FUNCTION_BLOCK MACH_CTL (* Cycle Control for a Machine with Fixed Tool *)
  (* Standard: 61499-1; Classification: Simulation; ApplicationDomain: Machining; Function: Drilling *)
  (* Version 0.2, 2004-10-20, JHC, Rockwell Automation, Changed algorithm to LD to recover from retracting fault. *)
  (* Version 0.1, 2004-04-05, JHC, Rockwell Automation, Corrected transition SPIN -> ADV *)
  (* Version 0.0, 2002-10-03, JHC, Rockwell Automation, Modified from DRILL_CTL. *)
  (* Compiler header: package fb.rt.mach; *)
  (* Compiler Java Sun JDK 1.4.2 *)
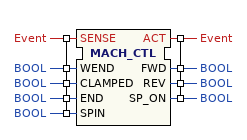
  EVENT_INPUT
    SENSE WITH WEND, CLAMPED, END, SPIN; (* Sensor data change *)
  END_EVENT
  EVENT_OUTPUT
    ACT WITH FWD, REV, SP_ON; (* Actuator output change *)
  END_EVENT
  VAR_INPUT
    WEND : BOOL; (* Workpiece present for machining *)
    CLAMPED : BOOL; (* Workpiece clamped *)
    END : BOOL; (* Machine at END position *)
    SPIN : BOOL; (* Spindle at operating speed *)
  END_VAR
  VAR_OUTPUT
    FWD : BOOL; (* Advance machine *)
    REV : BOOL; (* Retract machine *)
    SP_ON : BOOL; (* Spindle motor *)
  END_VAR
  VAR
    MACHINED : BOOL; (* Workpiece is machined *)
  END_VAR
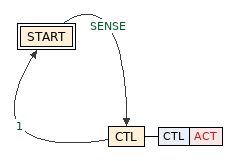
  EC_STATES
    START; (* Initial State *)
    CTL : CTL -> ACT; (* Execute Control Algorithm *)
  END_STATES
  EC_TRANSITIONS
    START TO CTL := SENSE;
    CTL TO START := 1;
  END_TRANSITIONS
  ALGORITHM CTL IN LD:
    SP_ON := CLAMPED;
    MACHINED := END MACHINED | CLAMPED &;
    FWD := SPIN WEND & MACHINED ! &;
    REV := FWD !;
  END_ALGORITHM
END_FUNCTION_BLOCK
